// TIA Portal V19 export
FUNCTION "FC_OUTPUT" : Void   // FC211, STL
TITLE = Schreiben der physikalischen Ausgänge
{ S7_Optimized_Access := 'FALSE' }
AUTHOR : RE
// stored: AutoNumber false
   VAR_TEMP
      Frg_Heben_li : Bool;
      Frg_Heben_re : Bool;
      Frg_Senken_li : Bool;
      Frg_Senken_re : Bool;
      Returnwert : Int;   // Rückgabewert SFC
      RetVal : Int;
   END_VAR
BEGIN

NETWORK
TITLE = Ausgabe
// Lampen

      A     "DB_ANLAGE".BA.Simulation;
      BEC;
//Warnung
      A     "DB_Alarme".Lampe_Gelb;
      O     "DB_ANLAGE".IN.Lamp_Test;
      =     "A_Mld_Wrn";
      =     "A_Mld_Wrn(2)";
      =     "A_Mld_Wrn_Geb.G";
// Störung
      A     "DB_Alarme".Lampe_Rot;
      O     "DB_ANLAGE".IN.Lamp_Test;
      =     "A_Mld_Al";
      =     "A_Mld_Al(2)";
      =     "A_Mld_Al_Geb.G";
//Hupe
      A     "DB_ANLAGE".OUT.Stoerung_Aku;
      =     "A_Hupe";
      =     "A_Hupe(2)";
      =     "A_Hupe_Geb.G";

//Fertigmeldung 1 WT will raus: CMD = 25
      L     "DB_WT1".akt_CMD;
      L     25;
      ==I;
      A     "DB_POS".POS["DB_WT1".POS].fertig;
      O(;
      L     "DB_WT2".akt_CMD;
      ==I;
      A     "DB_POS".POS["DB_WT2".POS].fertig;
      );
      O(;
      L     "DB_WT3".akt_CMD;
      L     25;
      ==I;
      A     "DB_POS".POS["DB_WT3".POS].fertig;
      );
      O(;
      L     "DB_WT4".akt_CMD;
      ==I;
      A     "DB_POS".POS["DB_WT4".POS].fertig;
      );
      O(;
      L     "DB_WT5".akt_CMD;
      L     25;
      ==I;
      A     "DB_POS".POS["DB_WT5".POS].fertig;
      );
      O(;
      L     "DB_WT6".akt_CMD;
      ==I;
      A     "DB_POS".POS["DB_WT6".POS].fertig;
      );
      O(;
      L     "DB_WT7".akt_CMD;
      L     25;
      ==I;
      A     "DB_POS".POS["DB_WT7".POS].fertig;
      );
      O(;
      L     "DB_WT8".akt_CMD;
      ==I;
      A     "DB_POS".POS["DB_WT8".POS].fertig;
      );
      O(;
      L     "DB_WT9".akt_CMD;
      L     25;
      ==I;
      A     "DB_POS".POS["DB_WT9".POS].fertig;
      );
      O(;
      L     "DB_WT10".akt_CMD;
      ==I;
      A     "DB_POS".POS["DB_WT10".POS].fertig;
      );
      O(;
      L     "DB_WT11".akt_CMD;
      L     25;
      ==I;
      A     "DB_POS".POS["DB_WT11".POS].fertig;
      );
      O(;
      L     "DB_WT12".akt_CMD;
      ==I;
      A     "DB_POS".POS["DB_WT12".POS].fertig;
      );
      A     "Clock_1Hz";
      O     "DI_FW_Auftrag_DB".Frg_Ausfahrt;
      O     "DB_ANLAGE".IN.Lamp_Test;
      =     "A_Mld_fertig";
      =     "A_Mld_fertig(2)";
      =     "A_Mld_fertig_Geb.G";

      A     "DB_ANLAGE".OUT.Fehler_Quitt;
      O     "DB_ANLAGE".IN.Lamp_Test;
      =     "A_LED_Q_Err";
      L     3;
      JC    LED;
      L     0;
LED:  T     "MobilePanel".Drucktaster_K2_LED;

      AN    "DB_PNOZ_IN_Out".In.PNOZ_OK;
      =     "A_LED_Q_NH";

// Meldung Automatik
      A     "DB_ANLAGE".OUT.MD_Auto;
      O     "DB_ANLAGE".IN.Lamp_Test;
      =     "A_Mld_Automatik";
      =     "A_Mld_Automatik(2)";
      =     "A_Mld_Automatik_Geb.G";

// Turmleuchte Tür
      AN    "E_Wrn_Gas_ok";
      =     "A_TL_T_Vorarlarm_Gas";
      =     "A_TL_T_Vorarlarm_Gas(2)";

      AN    "E_Al_Gas_ok";
      =     "A_TL_T_Hauptalarm_Gas";
      =     "A_TL_T_Hauptalarm_Gas(2)";

      AN    "E_Al_Gas_ok";
      =     "A_TL_T_Hupe";
      =     "A_TL_T_Hupe(2)";

// Koppelsignale
// --> AWA
      SET;
      =     "A_KS_in_Betrieb";
// --> Wäscher
      AN    "E_Niv_max_CM05.BL01";
      A     "E_Niv_Uel_CM05.BL12";
      =     "A_KS_CM05_nicht_Voll";

// Werkschutz
// 14x Leckage
      A     "FP_CM02.GP04".Mld.Leckage;
      O     "Pu_CL01.GP08".Mld.Leckage;
      O     "Pu_CL02.GP09".Mld.Leckage;
      O     "Pu_GP01.GP12".Mld.Leckage;
      O     "Pu_GP02.GP07".Mld.Leckage;
      O     "Pu_GP01.GP13".Mld.Leckage_Pumpe;
      O     "Pu_GP01.GP13".Mld.Leckage_PFA_Uebergang;
      O     "Pu_GP01.GP13".Mld.Leckage_Doppelrohr;
      O     "Pu_GP01.GP13".Mld.Leckage_Uml_Tunnel;
      O     "Pu_GP02.GP10".Mld.Leckage_Pumpe;
      O     "Pu_GP02.GP10".Mld.Leckage_PFA_Uebergang;
      ON    "E_LS_GP02.BL26";
      O     "Pu_GP02.GP10".Mld.Leckage_Doppelschlauch;
      ON    "E_LS_GP02.BL33";
      =     "A_Mld_WS_Leckage";
// 3x Überlauf
      A     "UP_CM01.GP02".Mld.Niv_Ueberlauf;
      O     "UP_CM02.GP05".Mld.Niv_Ueberlauf;
      O     "Pu_CM05.GP11_DB".Mld."Uel_CM05.BL05";
      =     "A_Mld_WS_Ueberlauf";

      A     "DB_Alarme".Lampe_Rot;
      =     "A_Mld_WS_SSt";

// LED Türen
      AN    "DB_PNOZ_IN_Out".In.Tuer_VS_ok;
      A     "Clock_1Hz";
      =     "A_LED_Tuer_VS";

      AN    "DB_PNOZ_IN_Out".In.Tuer_RS_ok;
      A     "Clock_1Hz";
      =     "A_LED_Tuer_RS";


NETWORK
TITLE = FW
// Transportsystem
// Reparaturbetrieb
      A     "DB_ANLAGE".IN.Reparatur;
      A     "DB_ANLAGE".IN.BA_Tipp;
      =     "A_RepB";

//--------------------------
//FW1
//--------------------------
// FU Fahrt: FU[10]

      CALL  "FB_FU_OUT_TW", "DI_FU_Fahrt"
      ( Req_High       := "DI_FW_1".OUT.VOR,
        Req_Low        := "DI_FW_1".OUT.RUECK,
        Reglersperre   := "FU_In_Out".FU[10].PA.Steuerwort.RegSp,
        Freigabe_Stopp := "FU_In_Out".FU[10].PA.Steuerwort.FrgStop,
        Freigabe_Halt  := "FU_In_Out".FU[10].PA.Steuerwort.FrgHalt,
        Break_ok       := "DI_FW_POS_1".IN.Break_on,
        SollSpeed      := "DI_FW_POS_1".OUT.SollSpeed,
        Ist_Speed      := "DI_FW_POS_1".IN.IstSpeed,
        PAW_Speed      := "FU_In_Out".FU[10].PA.Speed,
        PEW_Speed      := "FU_In_Out".FU[10].PE.Speed
      );

      A     "DI_FW_1".OUT.VOR;
      O     "DI_FW_1".OUT.RUECK;
      =     "A_Frg_FU_Fahrt";

// FU Hub links: FU[11]
      A     "DI_FW_1".OUT.HEBEN_li;
      =     "A_Heb_li";
      A     "DI_FW_1".OUT.SENKEN_li;
      =     "A_Snk_li";

      A     "DI_FW_1".OUT.HEBEN_li;
      A     "A_RepB";
      O     "E_Frg_Heb_li";
      =     #Frg_Heben_li;

      A     "DI_FW_1".OUT.SENKEN_li;
      A     "A_RepB";
      O     "E_Frg_Snk_li";
      =     #Frg_Senken_li;

      CALL  "FB_FU_OUT_TW", "DI_FU_Hub_links"
      ( Req_High       := #Frg_Heben_li,
        Req_Low        := #Frg_Senken_li,
        Reglersperre   := "FU_In_Out".FU[11].PA.Steuerwort.RegSp,
        Freigabe_Stopp := "FU_In_Out".FU[11].PA.Steuerwort.FrgStop,
        Freigabe_Halt  := "FU_In_Out".FU[11].PA.Steuerwort.FrgHalt,
        Break_ok       := "DI_FW_HUB_links".IN.Break_on,
        SollSpeed      := "DI_FW_HUB_links".OUT.SollSpeed,
        Ist_Speed      := "DI_FW_HUB_links".IN.IstSpeed,
        PAW_Speed      := "FU_In_Out".FU[11].PA.Speed,
        PEW_Speed      := "FU_In_Out".FU[11].PE.Speed
      );

      A     "DI_FW_1".OUT.HEBEN_li;
      O     "DI_FW_1".OUT.SENKEN_li;
      =     "A_Frg_FU_Hub_li";

      A     "DI_FW_1".ZST.Tipp;
      A     "DI_FW_1".ZST.BEREIT;
      A     "DI_FW_1".ZST.Unten_li;
      A     "T_ErrQuitt";
      =     "A_WZ_Tara_li_1";
      =     "A_WZ_Tara_li_2";
      =     "A_WZ_Tara_li_3";
      =     "A_WZ_Tara_li_4";

// FU Hub rechts: FU[12]
      A     "DI_FW_1".OUT.HEBEN_re;
      =     "A_Heb_re";
      A     "DI_FW_1".OUT.SENKEN_re;
      =     "A_Snk_re";

      A     "DI_FW_1".OUT.HEBEN_re;
      A     "A_RepB";
      O     "E_Frg_Heb_re";
      =     #Frg_Heben_re;

      A     "DI_FW_1".OUT.SENKEN_re;
      A     "A_RepB";
      O     "E_Frg_Snk_re";
      =     #Frg_Senken_re;

      CALL  "FB_FU_OUT_TW", "DI_FU_Hub_rechts"
      ( Req_High       := #Frg_Heben_re,
        Req_Low        := #Frg_Senken_re,
        Reglersperre   := "FU_In_Out".FU[12].PA.Steuerwort.RegSp,
        Freigabe_Stopp := "FU_In_Out".FU[12].PA.Steuerwort.FrgStop,
        Freigabe_Halt  := "FU_In_Out".FU[12].PA.Steuerwort.FrgHalt,
        Break_ok       := "DI_FW_HUB_rechts".IN.Break_on,
        SollSpeed      := "DI_FW_HUB_rechts".OUT.SollSpeed,
        Ist_Speed      := "DI_FW_HUB_rechts".IN.IstSpeed,
        PAW_Speed      := "FU_In_Out".FU[12].PA.Speed,
        PEW_Speed      := "FU_In_Out".FU[12].PE.Speed
      );

      A     "DI_FW_1".OUT.HEBEN_re;
      O     "DI_FW_1".OUT.SENKEN_re;
      =     "A_Frg_FU_Hub_re";


      A     "DI_FW_1".ZST.Tipp;
      A     "DI_FW_1".ZST.BEREIT;
      A     "DI_FW_1".ZST.Unten_re;
      A     "T_ErrQuitt";
      =     "A_WZ_Tara_re_1";
      =     "A_WZ_Tara_re_2";
      =     "A_WZ_Tara_re_3";
      =     "A_WZ_Tara_re_4";


NETWORK
TITLE = Be- und Entladestände (QF1 / QF2)
// WR02/03
// QF 1 FU[8]

      CALL  "FB_FU_OUT_TW", "DI_FU_WR02"
      ( Req_High       := "DI_QF_WR02_03".Out.WR02_einfahren,
        Req_Low        := "DI_QF_WR02_03".Out.WR02_ausfahren,
        Reglersperre   := "FU_In_Out".FU[8].PA.Steuerwort.RegSp,
        Freigabe_Stopp := "FU_In_Out".FU[8].PA.Steuerwort.FrgStop,
        Freigabe_Halt  := "FU_In_Out".FU[8].PA.Steuerwort.FrgHalt,
        Break_ok       := ,
        SollSpeed      := "DI_QF_WR02_03".Out.Soll_speed_WR02,
        Ist_Speed      := "DI_QF_WR02_03".In.FU_speed_WR02,
        PAW_Speed      := "FU_In_Out".FU[8].PA.Speed,
        PEW_Speed      := "FU_In_Out".FU[8].PE.Speed
      );

      A     "DI_QF_WR02_03".Out.WR02_einfahren;
      O     "DI_QF_WR02_03".Out.WR02_ausfahren;
      =     "A_Frg_FU_QF_WR02";

// QF 2 FU[9]

      CALL  "FB_FU_OUT_TW", "DI_FU_WR03"
      ( Req_High       := "DI_QF_WR02_03".Out.WR03_einfahren,
        Req_Low        := "DI_QF_WR02_03".Out.WR03_ausfahren,
        Reglersperre   := "FU_In_Out".FU[9].PA.Steuerwort.RegSp,
        Freigabe_Stopp := "FU_In_Out".FU[9].PA.Steuerwort.FrgStop,
        Freigabe_Halt  := "FU_In_Out".FU[9].PA.Steuerwort.FrgHalt,
        Break_ok       := ,
        SollSpeed      := "DI_QF_WR02_03".Out.Soll_speed_WR03,
        Ist_Speed      := "DI_QF_WR02_03".In.FU_speed_WR03,
        PAW_Speed      := "FU_In_Out".FU[9].PA.Speed,
        PEW_Speed      := "FU_In_Out".FU[9].PE.Speed
      );

      A     "DI_QF_WR02_03".Out.WR03_einfahren;
      O     "DI_QF_WR02_03".Out.WR03_ausfahren;
      =     "A_Frg_FU_QF_WR03";


NETWORK
TITLE = 
// Ausgänge
      CALL  "Output_Peripherie";

END_FUNCTION
